// SIMATIC STEP 7 (V5.x) project Starting
// CPU: CPU 313C
// station: Hardware
// station: SIMATIC 300(1)
// station: P_ADR_BUS
// station: P_ADR_BUS
// station: Configuration
// station: SIMATIC PC Station(1)
// program: S7 Program(1)

SYMBOL_TABLE
"start"	I 0.0	BOOL
"stop"	I 0.1	BOOL
END_SYMBOL_TABLE

FUNCTION_BLOCK FB 1
VERSION : 0.1
BEGIN
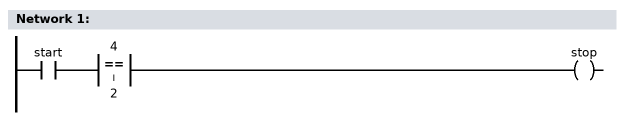
NETWORK
TITLE =
      A     "start";
      A(;
      L     4;
      L     2;
      ==I;
      );
      =     "stop";
END_FUNCTION_BLOCK

FUNCTION_BLOCK FB 2
VERSION : 0.1
BEGIN
// (block stored without names or comments; labels and parameter names are numbered)
END_FUNCTION_BLOCK

FUNCTION_BLOCK FB 3
VERSION : 0.1
BEGIN
// body was compiled from an S7-GRAPH chart; compiled code not shown
END_FUNCTION_BLOCK

ORGANIZATION_BLOCK OB 1
TITLE = "Main Program Sweep (Cycle)"
VERSION : 0.1
VAR_TEMP
  OB1_EV_CLASS : BYTE ;	//Bits 0-3 = 1 (Coming event), Bits 4-7 = 1 (Event class 1)
  OB1_SCAN_1 : BYTE ;	//1 (Cold restart scan 1 of OB 1), 3 (Scan 2-n of OB 1)
  OB1_PRIORITY : BYTE ;	//Priority of OB Execution
  OB1_OB_NUMBR : BYTE ;	//1 (Organization block 1, OB1)
  OB1_RESERVED_1 : BYTE ;	//Reserved for system
  OB1_RESERVED_2 : BYTE ;	//Reserved for system
  OB1_PREV_CYCLE : INT ;	//Cycle time of previous OB1 scan (milliseconds)
  OB1_MIN_CYCLE : INT ;	//Minimum cycle time of OB1 (milliseconds)
  OB1_MAX_CYCLE : INT ;	//Maximum cycle time of OB1 (milliseconds)
  OB1_DATE_TIME : DATE_AND_TIME ;	//Date and time OB1 started
END_VAR
BEGIN
// (block stored without names or comments; labels and parameter names are numbered)
END_ORGANIZATION_BLOCK
